Yaskawa INFORM job: spike.jbi

/JOB
//NAME SPIKE
//POS
///NPOS 4,0,0,0,0,0
///TOOL 0
///POSTYPE PULSE
///PULSE
C00000=0.000,-20.000,30.000,0.000,50.000,0.000
C00001=30.000,10.000,15.000,20.000,40.000,-10.000
C00002=10.000,20.000,30.000,40.000,50.000,60.000
C00003=0.000,0.000,0.000,0.000,0.000,0.000
//INST
///DATE 2000/01/01 00:00
///COMM tesseract emitters
///ATTR SC,RW
///GROUP1 RB1
NOP
'generated by tesseract_robotics.emitters <VERSION>
'ir-digest: sha256:8bab6d617b4fce14e73d25463528676423b617d59758612a304b441724c17d74
'profiles-digest: sha256:f8bd52140a239581a6137e8fc4b5b2dbc42c250b5cb4ac8c433864c12ffaec58
'DO NOT EDIT - regenerate from the planning pipeline
MOVJ C00000 VJ=50.00
MOVJ C00001 VJ=50.00
MOVJ C00002 VJ=50.00
MOVJ C00003 VJ=50.00
END
